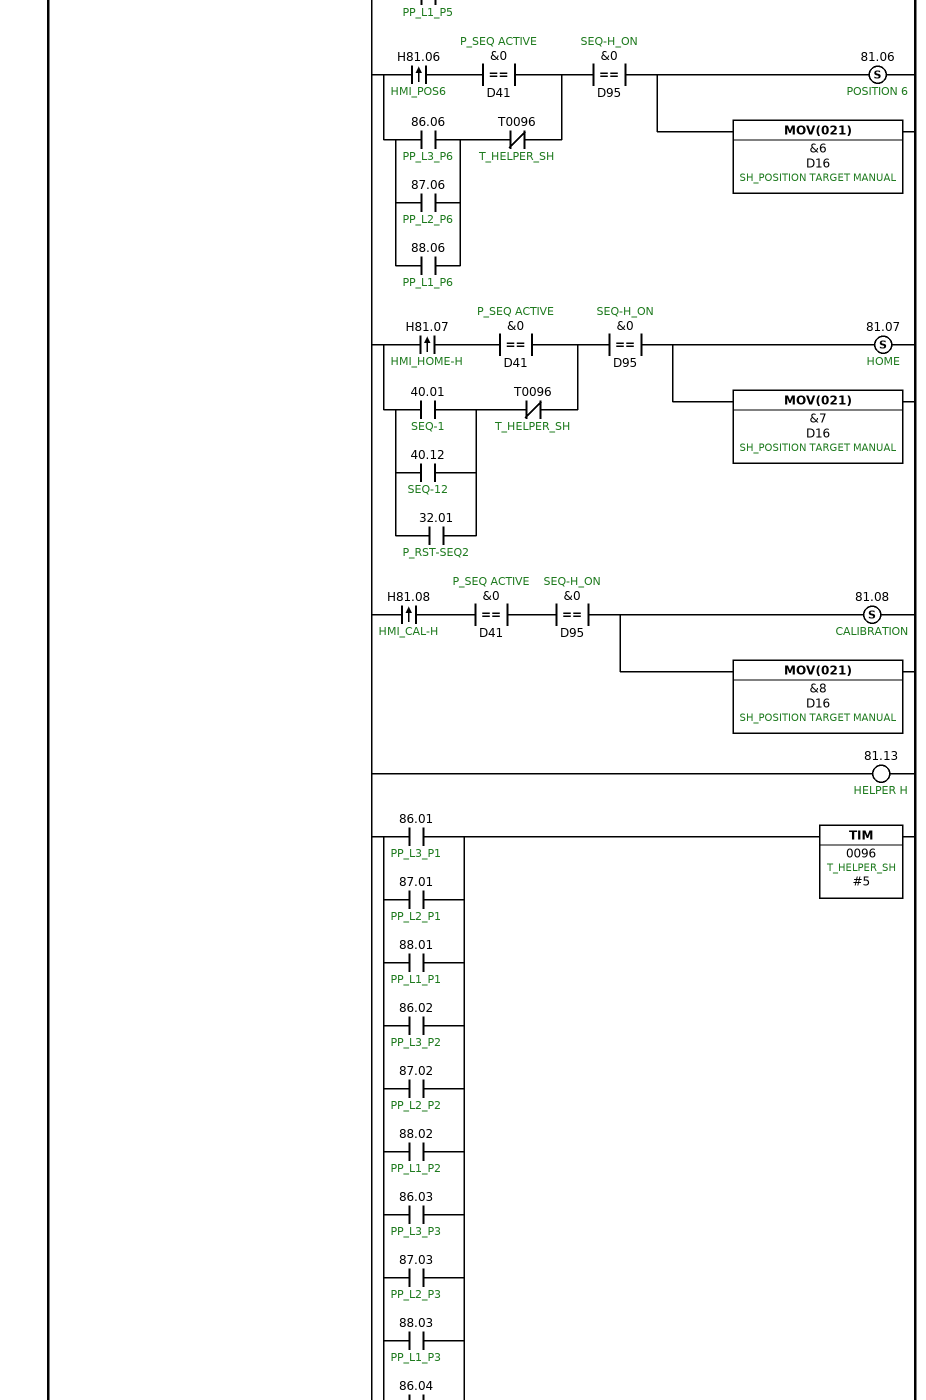
; [picture p24: NewProgram1 / SEQ_HORIZONTAL, rungs 1-1]

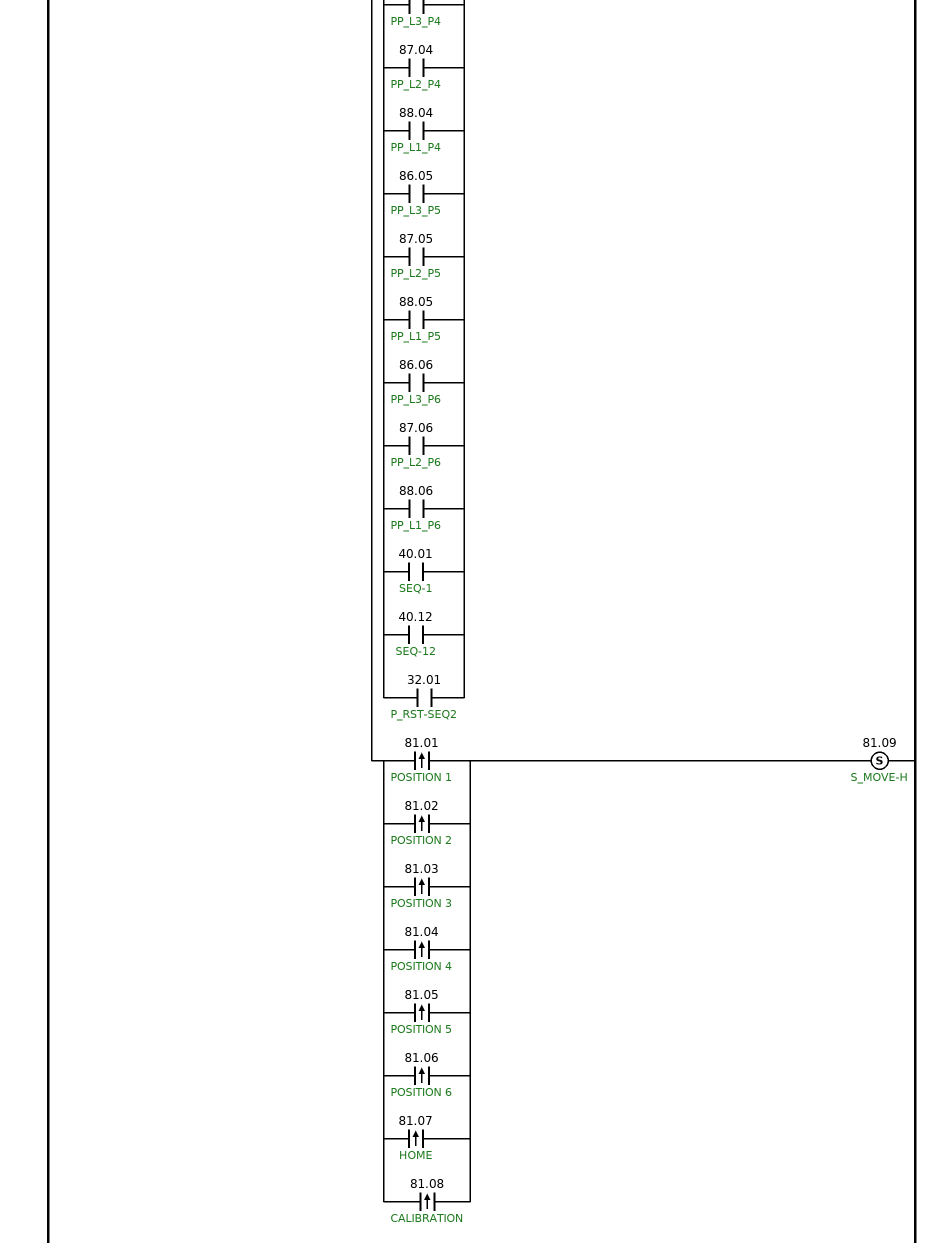
; rung 1: SET HORIZONTAL
LD P_On
LD=(300) &1 D41  ; P_SEQ ACTIVE
LD 40.01  ; SEQ-1
OR 40.08  ; SEQ-8
OR 40.12  ; SEQ-12
ANDLD
LD=(300) &1 D42  ; P_RST-SEQ_ACTIVE
AND 32.01  ; P_RST-SEQ2
ORLD
LD H30.00  ; HMI_C_MANUAL PAGE
AND=(300) &0 D41  ; P_SEQ ACTIVE
ORLD
ANDLD
OUT TR0
@LD H81.01  ; HMI_POS1
AND=(300) &0 D41  ; P_SEQ ACTIVE
LD 86.01  ; PP_L3_P1
OR 87.01  ; PP_L2_P1
OR 88.01  ; PP_L1_P1
ANDNOT T0096  ; T_HELPER_SH
ORLD
ANDLD
AND=(300) &0 D95  ; SEQ-H_ON
SET 81.01  ; POSITION 1
MOV(021) &1 D16  ; SH_POSITION TARGET MANUAL
LD TR0
@LD H81.02  ; HMI_POS2
AND=(300) &0 D41  ; P_SEQ ACTIVE
LD 86.02  ; PP_L3_P2
OR 87.02  ; PP_L2_P2
OR 88.02  ; PP_L1_P2
ANDNOT T0096  ; T_HELPER_SH
ORLD
ANDLD
AND=(300) &0 D95  ; SEQ-H_ON
SET 81.02  ; POSITION 2
MOV(021) &2 D16  ; SH_POSITION TARGET MANUAL
LD TR0
@LD H81.03  ; HMI_POS3
AND=(300) &0 D41  ; P_SEQ ACTIVE
LD 86.03  ; PP_L3_P3
OR 87.03  ; PP_L2_P3
OR 88.03  ; PP_L1_P3
ANDNOT T0096  ; T_HELPER_SH
ORLD
ANDLD
AND=(300) &0 D95  ; SEQ-H_ON
SET 81.03  ; POSITION 3
MOV(021) &3 D16  ; SH_POSITION TARGET MANUAL
LD TR0
@LD H81.04  ; HMI_POS4
AND=(300) &0 D41  ; P_SEQ ACTIVE
LD 86.04  ; PP_L3_P4
OR 87.04  ; PP_L2_P4
OR 88.04  ; PP_L1_P4
ANDNOT T0096  ; T_HELPER_SH
ORLD
ANDLD
AND=(300) &0 D95  ; SEQ-H_ON
SET 81.04  ; POSITION 4
MOV(021) &4 D16  ; SH_POSITION TARGET MANUAL
LD TR0
@LD H81.05  ; HMI_POS5
AND=(300) &0 D41  ; P_SEQ ACTIVE
LD 86.05  ; PP_L3_P5
OR 87.05  ; PP_L2_P5
OR 88.05  ; PP_L1_P5
ANDNOT T0096  ; T_HELPER_SH
ORLD
ANDLD
AND=(300) &0 D95  ; SEQ-H_ON
SET 81.05  ; POSITION 5
MOV(021) &5 D16  ; SH_POSITION TARGET MANUAL
LD TR0
@LD H81.06  ; HMI_POS6
AND=(300) &0 D41  ; P_SEQ ACTIVE
LD 86.06  ; PP_L3_P6
OR 87.06  ; PP_L2_P6
OR 88.06  ; PP_L1_P6
ANDNOT T0096  ; T_HELPER_SH
ORLD
ANDLD
AND=(300) &0 D95  ; SEQ-H_ON
SET 81.06  ; POSITION 6
MOV(021) &6 D16  ; SH_POSITION TARGET MANUAL
LD TR0
@LD H81.07  ; HMI_HOME-H
AND=(300) &0 D41  ; P_SEQ ACTIVE
LD 40.01  ; SEQ-1
OR 40.12  ; SEQ-12
OR 32.01  ; P_RST-SEQ2
ANDNOT T0096  ; T_HELPER_SH
ORLD
ANDLD
AND=(300) &0 D95  ; SEQ-H_ON
SET 81.07  ; HOME
MOV(021) &7 D16  ; SH_POSITION TARGET MANUAL
LD TR0
@AND H81.08  ; HMI_CAL-H
AND=(300) &0 D41  ; P_SEQ ACTIVE
AND=(300) &0 D95  ; SEQ-H_ON
SET 81.08  ; CALIBRATION
MOV(021) &8 D16  ; SH_POSITION TARGET MANUAL
LD TR0
OUT 81.13  ; HELPER H
LD 86.01  ; PP_L3_P1
OR 87.01  ; PP_L2_P1
OR 88.01  ; PP_L1_P1
OR 86.02  ; PP_L3_P2
OR 87.02  ; PP_L2_P2
OR 88.02  ; PP_L1_P2
OR 86.03  ; PP_L3_P3
OR 87.03  ; PP_L2_P3
OR 88.03  ; PP_L1_P3
OR 86.04  ; PP_L3_P4
OR 87.04  ; PP_L2_P4
OR 88.04  ; PP_L1_P4
OR 86.05  ; PP_L3_P5
OR 87.05  ; PP_L2_P5
OR 88.05  ; PP_L1_P5
OR 86.06  ; PP_L3_P6
OR 87.06  ; PP_L2_P6
OR 88.06  ; PP_L1_P6
OR 40.01  ; SEQ-1
OR 40.12  ; SEQ-12
OR 32.01  ; P_RST-SEQ2
ANDLD
TIM 0096 #5  ; T_HELPER_SH
LD TR0
@LD 81.01  ; POSITION 1
@OR 81.02  ; POSITION 2
@OR 81.03  ; POSITION 3
@OR 81.04  ; POSITION 4
@OR 81.05  ; POSITION 5
@OR 81.06  ; POSITION 6
@OR 81.07  ; HOME
@OR 81.08  ; CALIBRATION
ANDLD
SET 81.09  ; S_MOVE-H

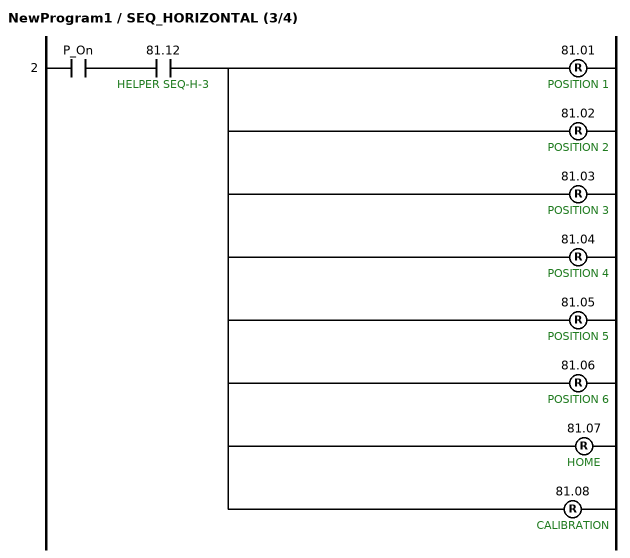
; rung 2
LD P_On
AND 81.12  ; HELPER SEQ-H-3
RSET 81.01  ; POSITION 1
RSET 81.02  ; POSITION 2
RSET 81.03  ; POSITION 3
RSET 81.04  ; POSITION 4
RSET 81.05  ; POSITION 5
RSET 81.06  ; POSITION 6
RSET 81.07  ; HOME
RSET 81.08  ; CALIBRATION

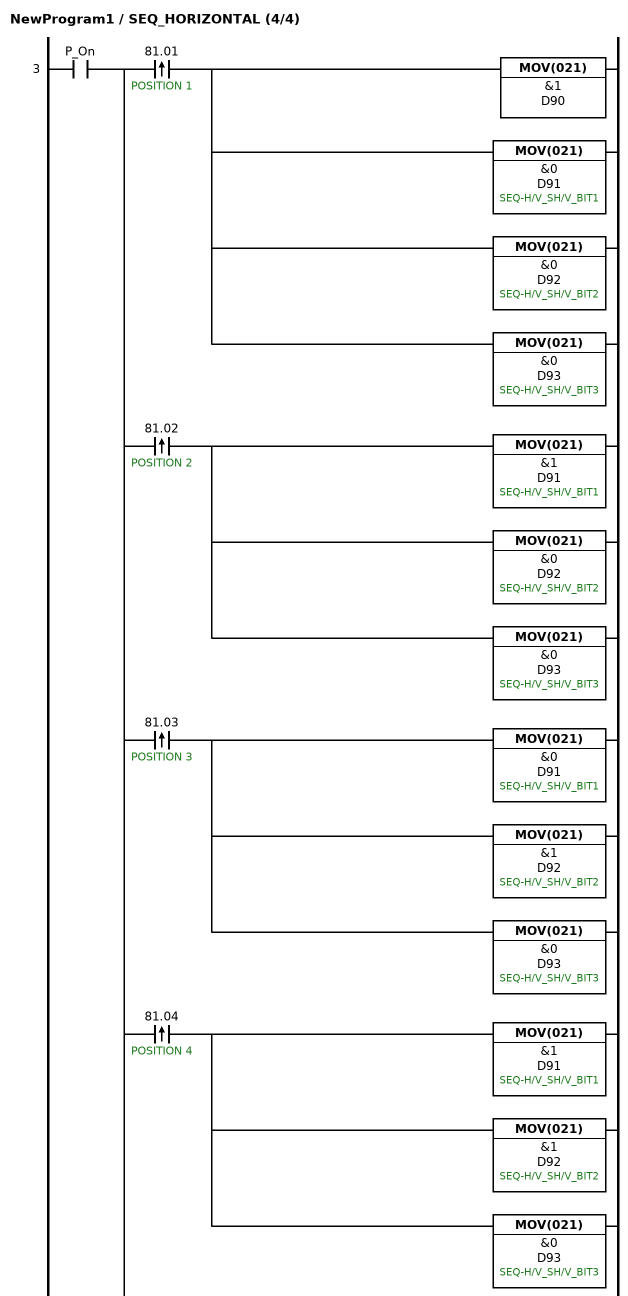

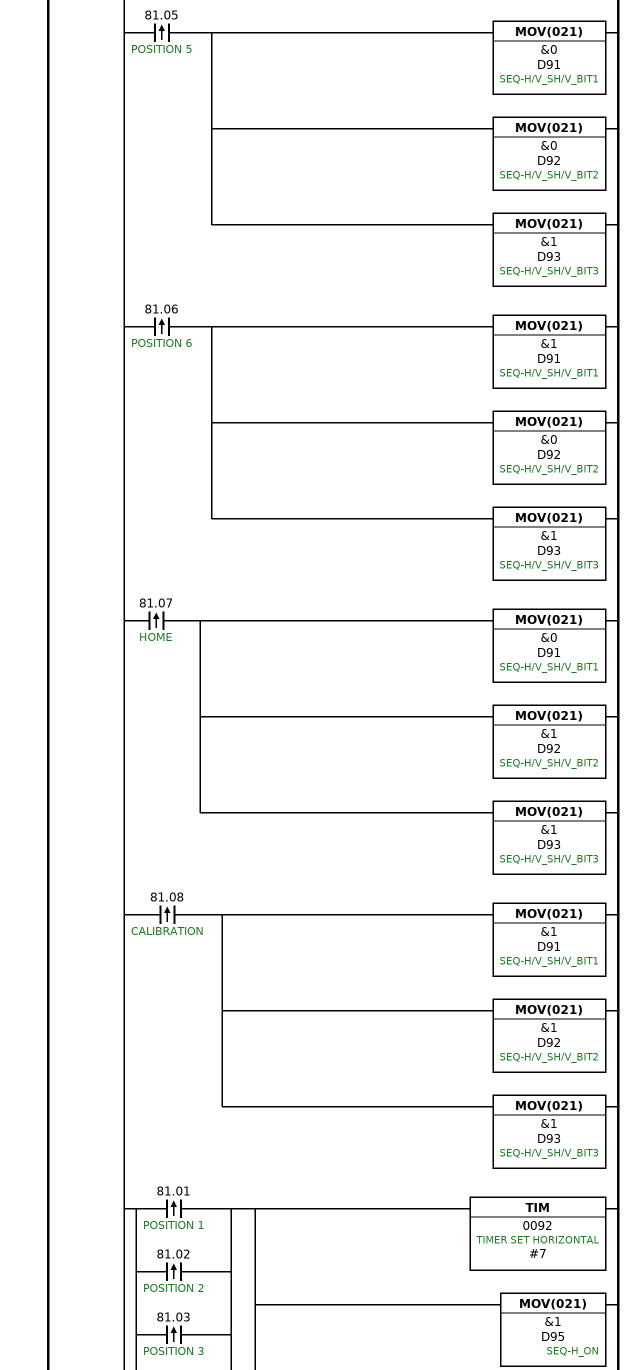

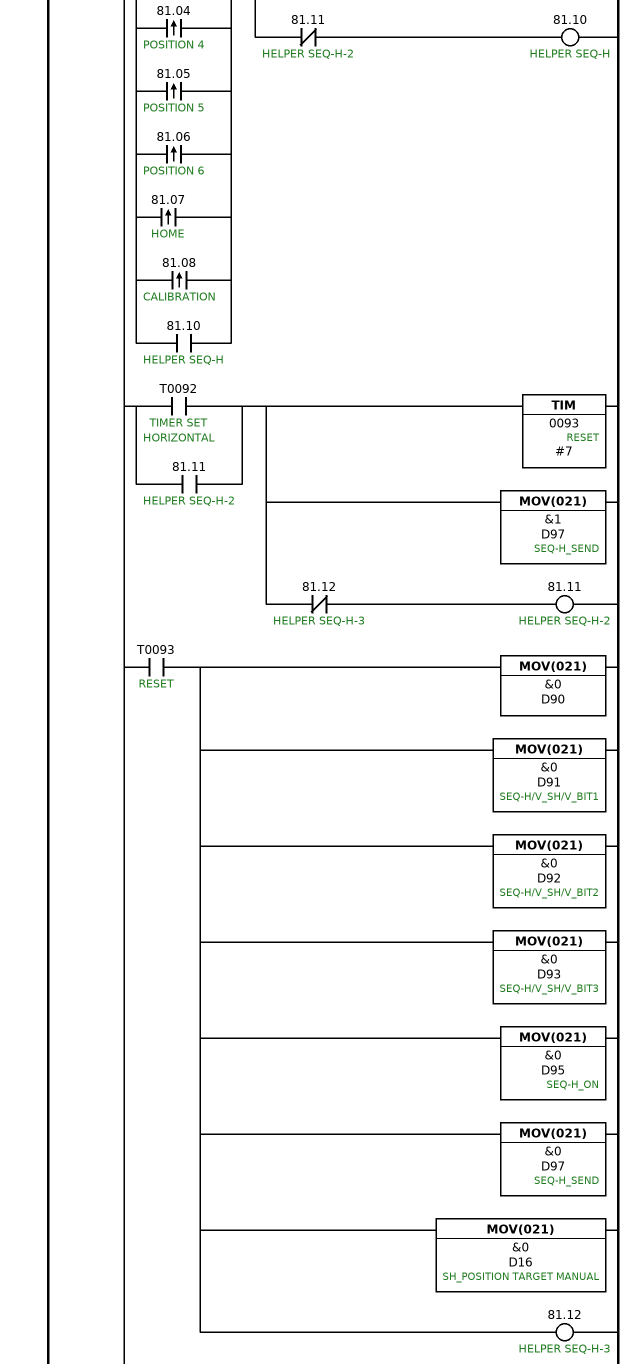

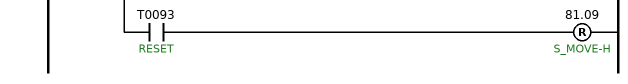
; rung 3
LD P_On
OUT TR0
@AND 81.01  ; POSITION 1
MOV(021) &1 D90
MOV(021) &0 D91  ; SEQ-H/V_SH/V_BIT1
MOV(021) &0 D92  ; SEQ-H/V_SH/V_BIT2
MOV(021) &0 D93  ; SEQ-H/V_SH/V_BIT3
LD TR0
@AND 81.02  ; POSITION 2
MOV(021) &1 D91  ; SEQ-H/V_SH/V_BIT1
MOV(021) &0 D92  ; SEQ-H/V_SH/V_BIT2
MOV(021) &0 D93  ; SEQ-H/V_SH/V_BIT3
LD TR0
@AND 81.03  ; POSITION 3
MOV(021) &0 D91  ; SEQ-H/V_SH/V_BIT1
MOV(021) &1 D92  ; SEQ-H/V_SH/V_BIT2
MOV(021) &0 D93  ; SEQ-H/V_SH/V_BIT3
LD TR0
@AND 81.04  ; POSITION 4
MOV(021) &1 D91  ; SEQ-H/V_SH/V_BIT1
MOV(021) &1 D92  ; SEQ-H/V_SH/V_BIT2
MOV(021) &0 D93  ; SEQ-H/V_SH/V_BIT3
LD TR0
@AND 81.05  ; POSITION 5
MOV(021) &0 D91  ; SEQ-H/V_SH/V_BIT1
MOV(021) &0 D92  ; SEQ-H/V_SH/V_BIT2
MOV(021) &1 D93  ; SEQ-H/V_SH/V_BIT3
LD TR0
@AND 81.06  ; POSITION 6
MOV(021) &1 D91  ; SEQ-H/V_SH/V_BIT1
MOV(021) &0 D92  ; SEQ-H/V_SH/V_BIT2
MOV(021) &1 D93  ; SEQ-H/V_SH/V_BIT3
LD TR0
@AND 81.07  ; HOME
MOV(021) &0 D91  ; SEQ-H/V_SH/V_BIT1
MOV(021) &1 D92  ; SEQ-H/V_SH/V_BIT2
MOV(021) &1 D93  ; SEQ-H/V_SH/V_BIT3
LD TR0
@AND 81.08  ; CALIBRATION
MOV(021) &1 D91  ; SEQ-H/V_SH/V_BIT1
MOV(021) &1 D92  ; SEQ-H/V_SH/V_BIT2
MOV(021) &1 D93  ; SEQ-H/V_SH/V_BIT3
LD TR0
@LD 81.01  ; POSITION 1
@OR 81.02  ; POSITION 2
@OR 81.03  ; POSITION 3
@OR 81.04  ; POSITION 4
@OR 81.05  ; POSITION 5
@OR 81.06  ; POSITION 6
@OR 81.07  ; HOME
@OR 81.08  ; CALIBRATION
OR 81.10  ; HELPER SEQ-H
ANDLD
TIM 0092 #7  ; TIMER SET HORIZONTAL
MOV(021) &1 D95  ; SEQ-H_ON
ANDNOT 81.11  ; HELPER SEQ-H-2
OUT 81.10  ; HELPER SEQ-H
LD TR0
LD T0092  ; TIMER SET HORIZONTAL
OR 81.11  ; HELPER SEQ-H-2
ANDLD
TIM 0093 #7  ; RESET
MOV(021) &1 D97  ; SEQ-H_SEND
ANDNOT 81.12  ; HELPER SEQ-H-3
OUT 81.11  ; HELPER SEQ-H-2
LD TR0
AND T0093  ; RESET
MOV(021) &0 D90
MOV(021) &0 D91  ; SEQ-H/V_SH/V_BIT1
MOV(021) &0 D92  ; SEQ-H/V_SH/V_BIT2
MOV(021) &0 D93  ; SEQ-H/V_SH/V_BIT3
MOV(021) &0 D95  ; SEQ-H_ON
MOV(021) &0 D97  ; SEQ-H_SEND
MOV(021) &0 D16  ; SH_POSITION TARGET MANUAL
OUT 81.12  ; HELPER SEQ-H-3
LD TR0
AND T0093  ; RESET
RSET 81.09  ; S_MOVE-H

### Section SEQ_VERTICAL

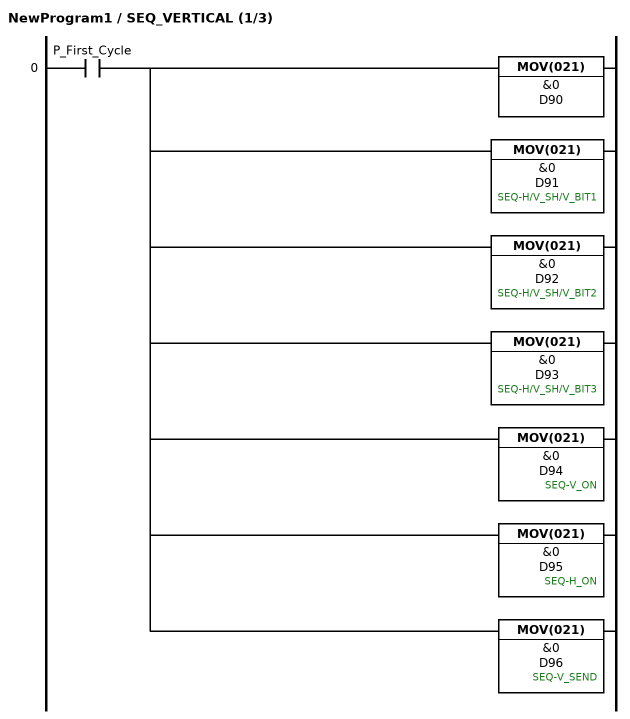
; rung 0
LD P_First_Cycle
MOV(021) &0 D90
MOV(021) &0 D91  ; SEQ-H/V_SH/V_BIT1
MOV(021) &0 D92  ; SEQ-H/V_SH/V_BIT2
MOV(021) &0 D93  ; SEQ-H/V_SH/V_BIT3
MOV(021) &0 D94  ; SEQ-V_ON
MOV(021) &0 D95  ; SEQ-H_ON
MOV(021) &0 D96  ; SEQ-V_SEND

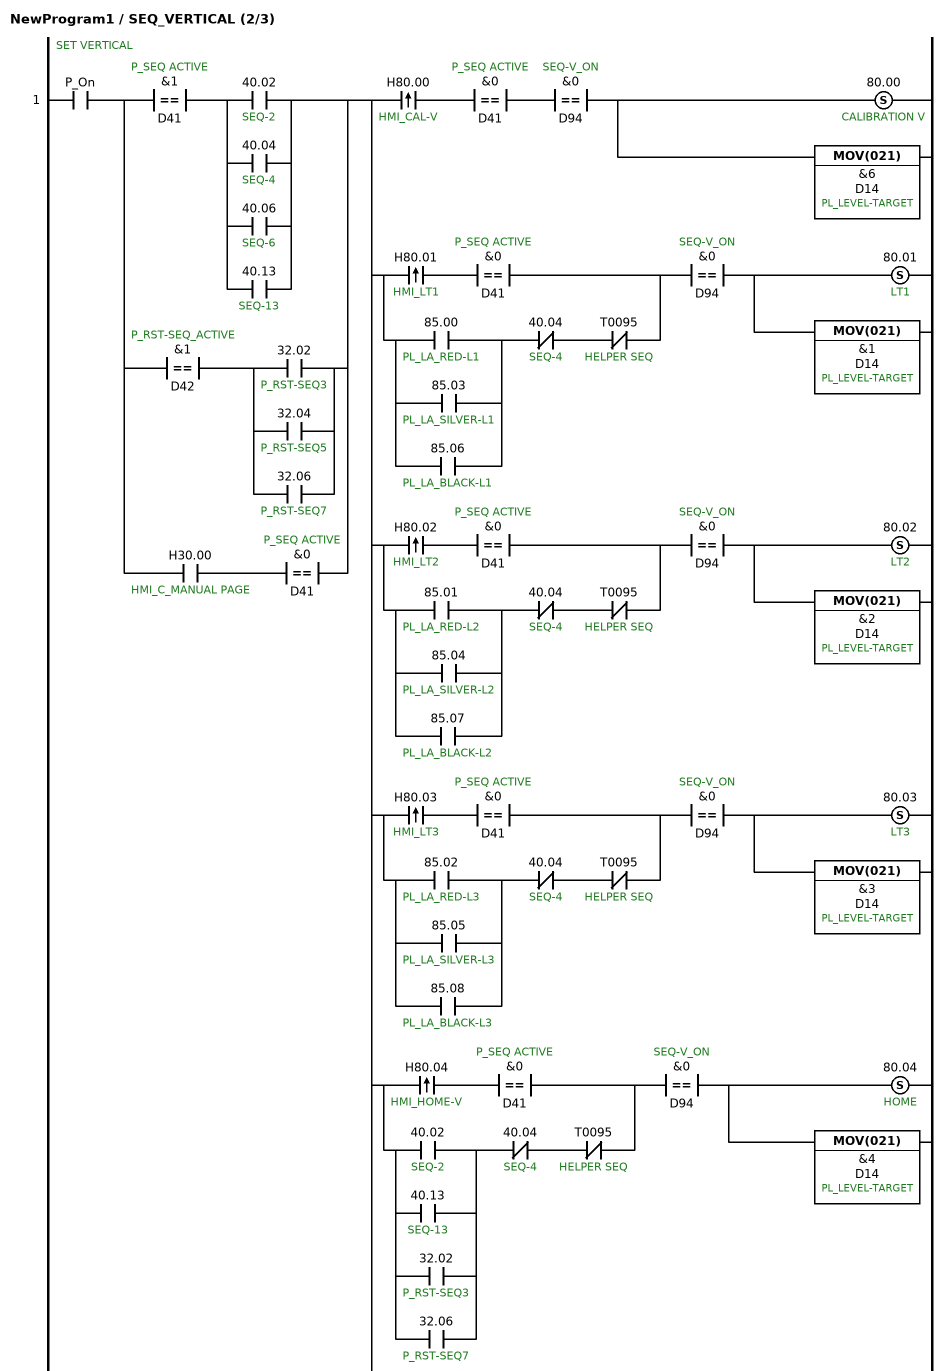

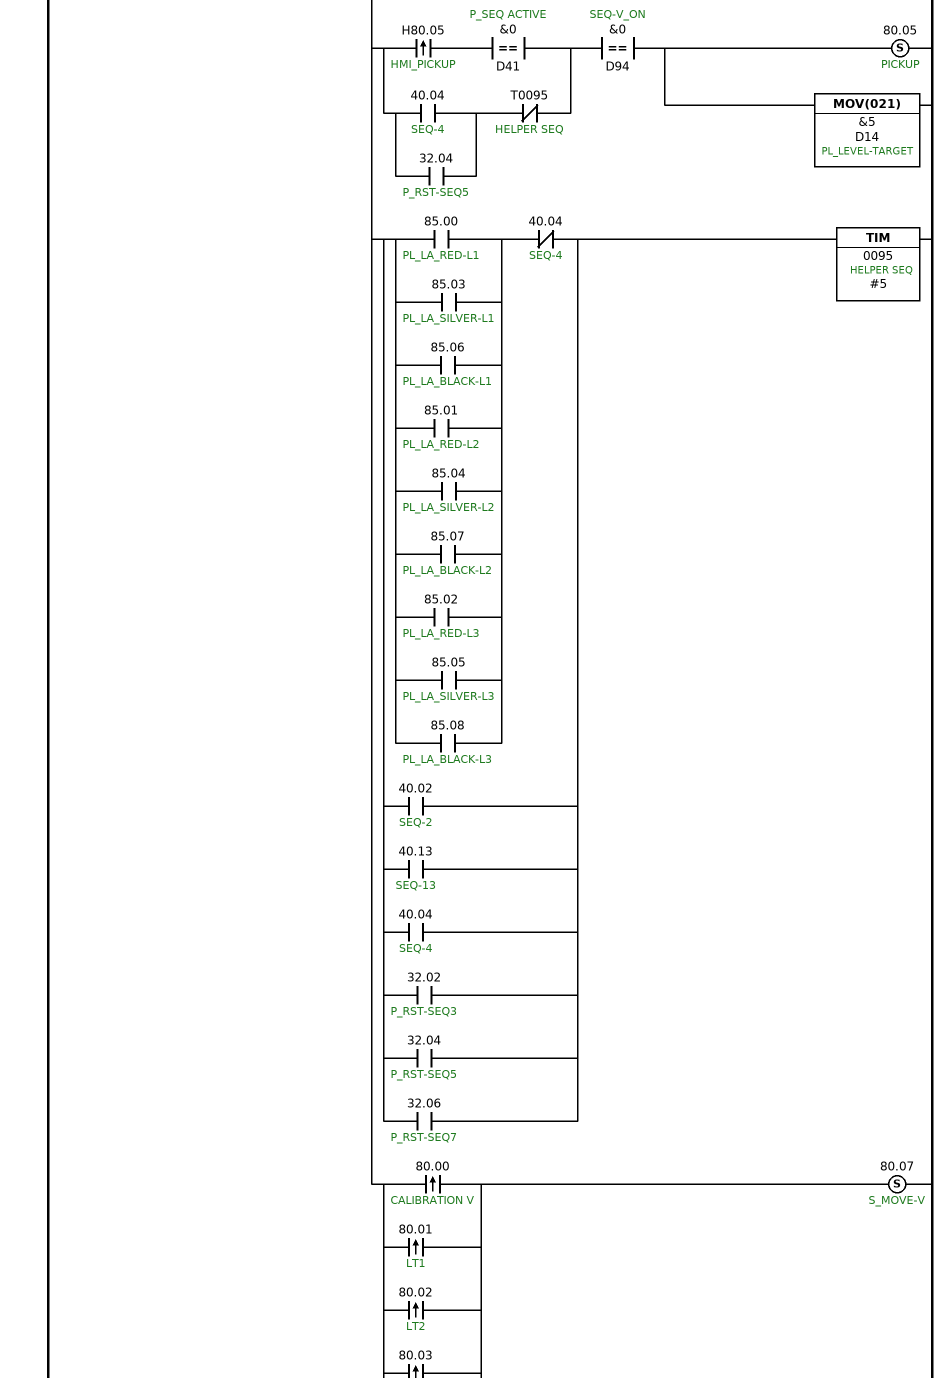

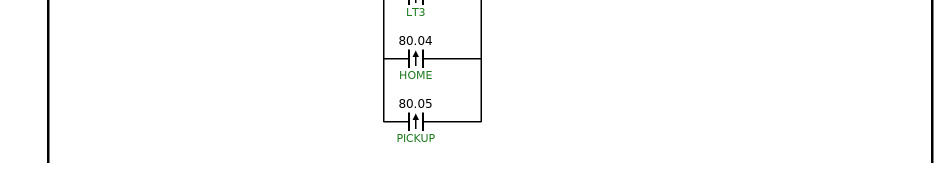
; rung 1: SET VERTICAL
LD P_On
LD=(300) &1 D41  ; P_SEQ ACTIVE
LD 40.02  ; SEQ-2
OR 40.04  ; SEQ-4
OR 40.06  ; SEQ-6
OR 40.13  ; SEQ-13
ANDLD
LD=(300) &1 D42  ; P_RST-SEQ_ACTIVE
LD 32.02  ; P_RST-SEQ3
OR 32.04  ; P_RST-SEQ5
OR 32.06  ; P_RST-SEQ7
ANDLD
ORLD
LD H30.00  ; HMI_C_MANUAL PAGE
AND=(300) &0 D41  ; P_SEQ ACTIVE
ORLD
ANDLD
OUT TR0
@AND H80.00  ; HMI_CAL-V
AND=(300) &0 D41  ; P_SEQ ACTIVE
AND=(300) &0 D94  ; SEQ-V_ON
SET 80.00  ; CALIBRATION V
MOV(021) &6 D14  ; PL_LEVEL-TARGET
LD TR0
@LD H80.01  ; HMI_LT1
AND=(300) &0 D41  ; P_SEQ ACTIVE
LD 85.00  ; PL_LA_RED-L1
OR 85.03  ; PL_LA_SILVER-L1
OR 85.06  ; PL_LA_BLACK-L1
ANDNOT 40.04  ; SEQ-4
ANDNOT T0095  ; HELPER SEQ
ORLD
ANDLD
AND=(300) &0 D94  ; SEQ-V_ON
SET 80.01  ; LT1
MOV(021) &1 D14  ; PL_LEVEL-TARGET
LD TR0
@LD H80.02  ; HMI_LT2
AND=(300) &0 D41  ; P_SEQ ACTIVE
LD 85.01  ; PL_LA_RED-L2
OR 85.04  ; PL_LA_SILVER-L2
OR 85.07  ; PL_LA_BLACK-L2
ANDNOT 40.04  ; SEQ-4
ANDNOT T0095  ; HELPER SEQ
ORLD
ANDLD
AND=(300) &0 D94  ; SEQ-V_ON
SET 80.02  ; LT2
MOV(021) &2 D14  ; PL_LEVEL-TARGET
LD TR0
@LD H80.03  ; HMI_LT3
AND=(300) &0 D41  ; P_SEQ ACTIVE
LD 85.02  ; PL_LA_RED-L3
OR 85.05  ; PL_LA_SILVER-L3
OR 85.08  ; PL_LA_BLACK-L3
ANDNOT 40.04  ; SEQ-4
ANDNOT T0095  ; HELPER SEQ
ORLD
ANDLD
AND=(300) &0 D94  ; SEQ-V_ON
SET 80.03  ; LT3
MOV(021) &3 D14  ; PL_LEVEL-TARGET
LD TR0
@LD H80.04  ; HMI_HOME-V
AND=(300) &0 D41  ; P_SEQ ACTIVE
LD 40.02  ; SEQ-2
OR 40.13  ; SEQ-13
OR 32.02  ; P_RST-SEQ3
OR 32.06  ; P_RST-SEQ7
ANDNOT 40.04  ; SEQ-4
ANDNOT T0095  ; HELPER SEQ
ORLD
ANDLD
AND=(300) &0 D94  ; SEQ-V_ON
SET 80.04  ; HOME
MOV(021) &4 D14  ; PL_LEVEL-TARGET
LD TR0
@LD H80.05  ; HMI_PICKUP
AND=(300) &0 D41  ; P_SEQ ACTIVE
LD 40.04  ; SEQ-4
OR 32.04  ; P_RST-SEQ5
ANDNOT T0095  ; HELPER SEQ
ORLD
ANDLD
AND=(300) &0 D94  ; SEQ-V_ON
SET 80.05  ; PICKUP
MOV(021) &5 D14  ; PL_LEVEL-TARGET
LD TR0
LD 85.00  ; PL_LA_RED-L1
OR 85.03  ; PL_LA_SILVER-L1
OR 85.06  ; PL_LA_BLACK-L1
OR 85.01  ; PL_LA_RED-L2
OR 85.04  ; PL_LA_SILVER-L2
OR 85.07  ; PL_LA_BLACK-L2
OR 85.02  ; PL_LA_RED-L3
OR 85.05  ; PL_LA_SILVER-L3
OR 85.08  ; PL_LA_BLACK-L3
ANDNOT 40.04  ; SEQ-4
OR 40.02  ; SEQ-2
OR 40.13  ; SEQ-13
OR 40.04  ; SEQ-4
OR 32.02  ; P_RST-SEQ3
OR 32.04  ; P_RST-SEQ5
OR 32.06  ; P_RST-SEQ7
ANDLD
TIM 0095 #5  ; HELPER SEQ
LD TR0
@LD 80.00  ; CALIBRATION V
@OR 80.01  ; LT1
@OR 80.02  ; LT2
@OR 80.03  ; LT3
@OR 80.04  ; HOME
@OR 80.05  ; PICKUP
ANDLD
SET 80.07  ; S_MOVE-V

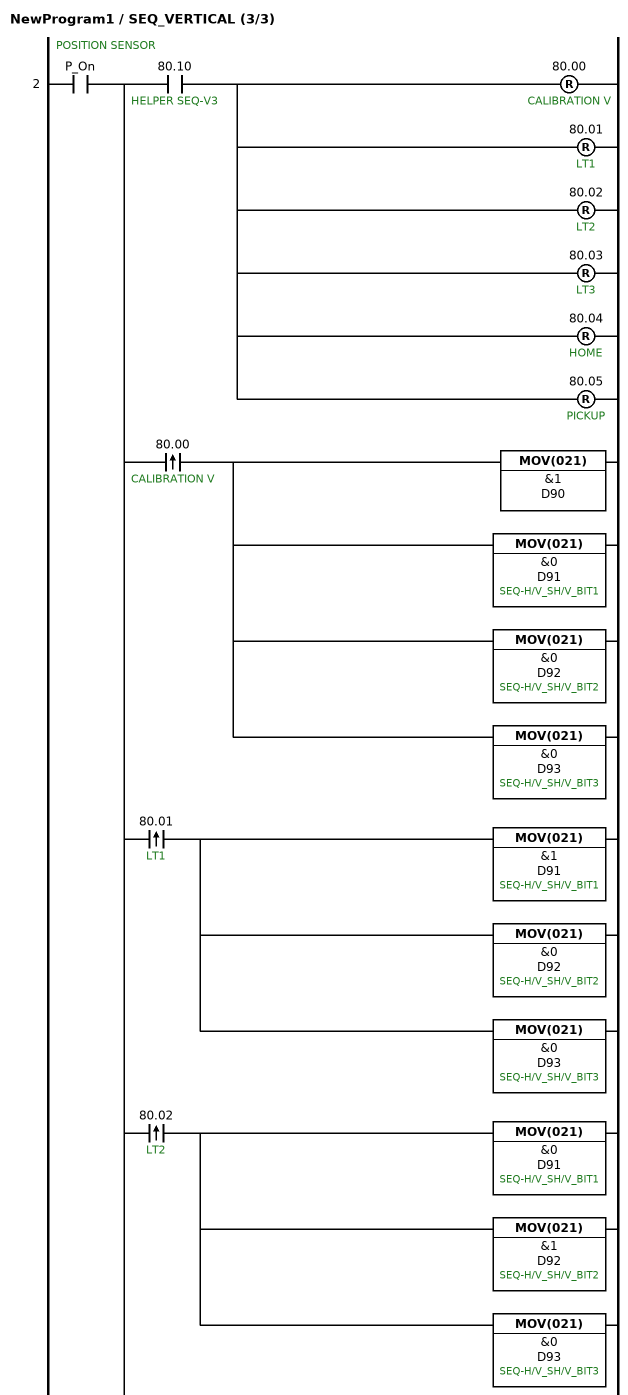

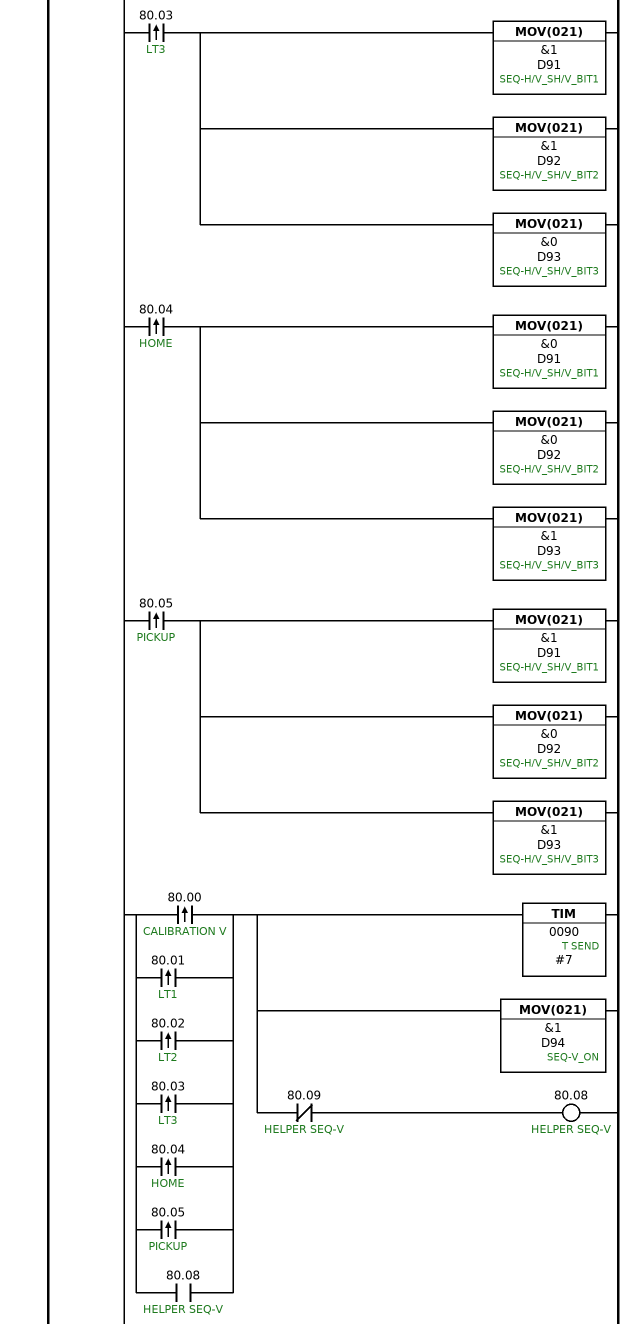

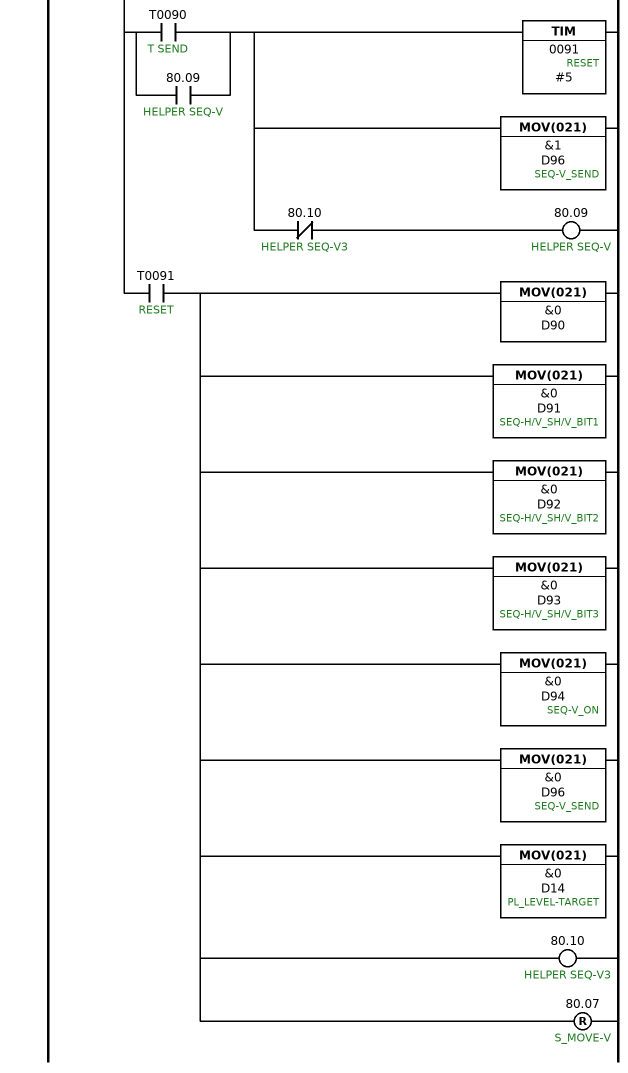
; rung 2: POSITION SENSOR
LD P_On
OUT TR0
AND 80.10  ; HELPER SEQ-V3
RSET 80.00  ; CALIBRATION V
RSET 80.01  ; LT1
RSET 80.02  ; LT2
RSET 80.03  ; LT3
RSET 80.04  ; HOME
RSET 80.05  ; PICKUP
LD TR0
@AND 80.00  ; CALIBRATION V
MOV(021) &1 D90
MOV(021) &0 D91  ; SEQ-H/V_SH/V_BIT1
MOV(021) &0 D92  ; SEQ-H/V_SH/V_BIT2
MOV(021) &0 D93  ; SEQ-H/V_SH/V_BIT3
LD TR0
@AND 80.01  ; LT1
MOV(021) &1 D91  ; SEQ-H/V_SH/V_BIT1
MOV(021) &0 D92  ; SEQ-H/V_SH/V_BIT2
MOV(021) &0 D93  ; SEQ-H/V_SH/V_BIT3
LD TR0
@AND 80.02  ; LT2
MOV(021) &0 D91  ; SEQ-H/V_SH/V_BIT1
MOV(021) &1 D92  ; SEQ-H/V_SH/V_BIT2
MOV(021) &0 D93  ; SEQ-H/V_SH/V_BIT3
LD TR0
@AND 80.03  ; LT3
MOV(021) &1 D91  ; SEQ-H/V_SH/V_BIT1
MOV(021) &1 D92  ; SEQ-H/V_SH/V_BIT2
MOV(021) &0 D93  ; SEQ-H/V_SH/V_BIT3
LD TR0
@AND 80.04  ; HOME
MOV(021) &0 D91  ; SEQ-H/V_SH/V_BIT1
MOV(021) &0 D92  ; SEQ-H/V_SH/V_BIT2
MOV(021) &1 D93  ; SEQ-H/V_SH/V_BIT3
LD TR0
@AND 80.05  ; PICKUP
MOV(021) &1 D91  ; SEQ-H/V_SH/V_BIT1
MOV(021) &0 D92  ; SEQ-H/V_SH/V_BIT2
MOV(021) &1 D93  ; SEQ-H/V_SH/V_BIT3
LD TR0
@LD 80.00  ; CALIBRATION V
@OR 80.01  ; LT1
@OR 80.02  ; LT2
@OR 80.03  ; LT3
@OR 80.04  ; HOME
@OR 80.05  ; PICKUP
OR 80.08  ; HELPER SEQ-V
ANDLD
TIM 0090 #7  ; T SEND
MOV(021) &1 D94  ; SEQ-V_ON
ANDNOT 80.09  ; HELPER SEQ-V
OUT 80.08  ; HELPER SEQ-V
LD TR0
LD T0090  ; T SEND
OR 80.09  ; HELPER SEQ-V
ANDLD
TIM 0091 #5  ; RESET
MOV(021) &1 D96  ; SEQ-V_SEND
ANDNOT 80.10  ; HELPER SEQ-V3
OUT 80.09  ; HELPER SEQ-V
LD TR0
AND T0091  ; RESET
MOV(021) &0 D90
MOV(021) &0 D91  ; SEQ-H/V_SH/V_BIT1
MOV(021) &0 D92  ; SEQ-H/V_SH/V_BIT2
MOV(021) &0 D93  ; SEQ-H/V_SH/V_BIT3
MOV(021) &0 D94  ; SEQ-V_ON
MOV(021) &0 D96  ; SEQ-V_SEND
MOV(021) &0 D14  ; PL_LEVEL-TARGET
OUT 80.10  ; HELPER SEQ-V3
RSET 80.07  ; S_MOVE-V

### Section SEQUENCE

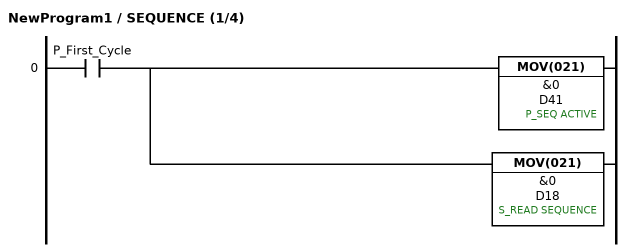
; rung 0
LD P_First_Cycle
MOV(021) &0 D41  ; P_SEQ ACTIVE
MOV(021) &0 D18  ; S_READ SEQUENCE

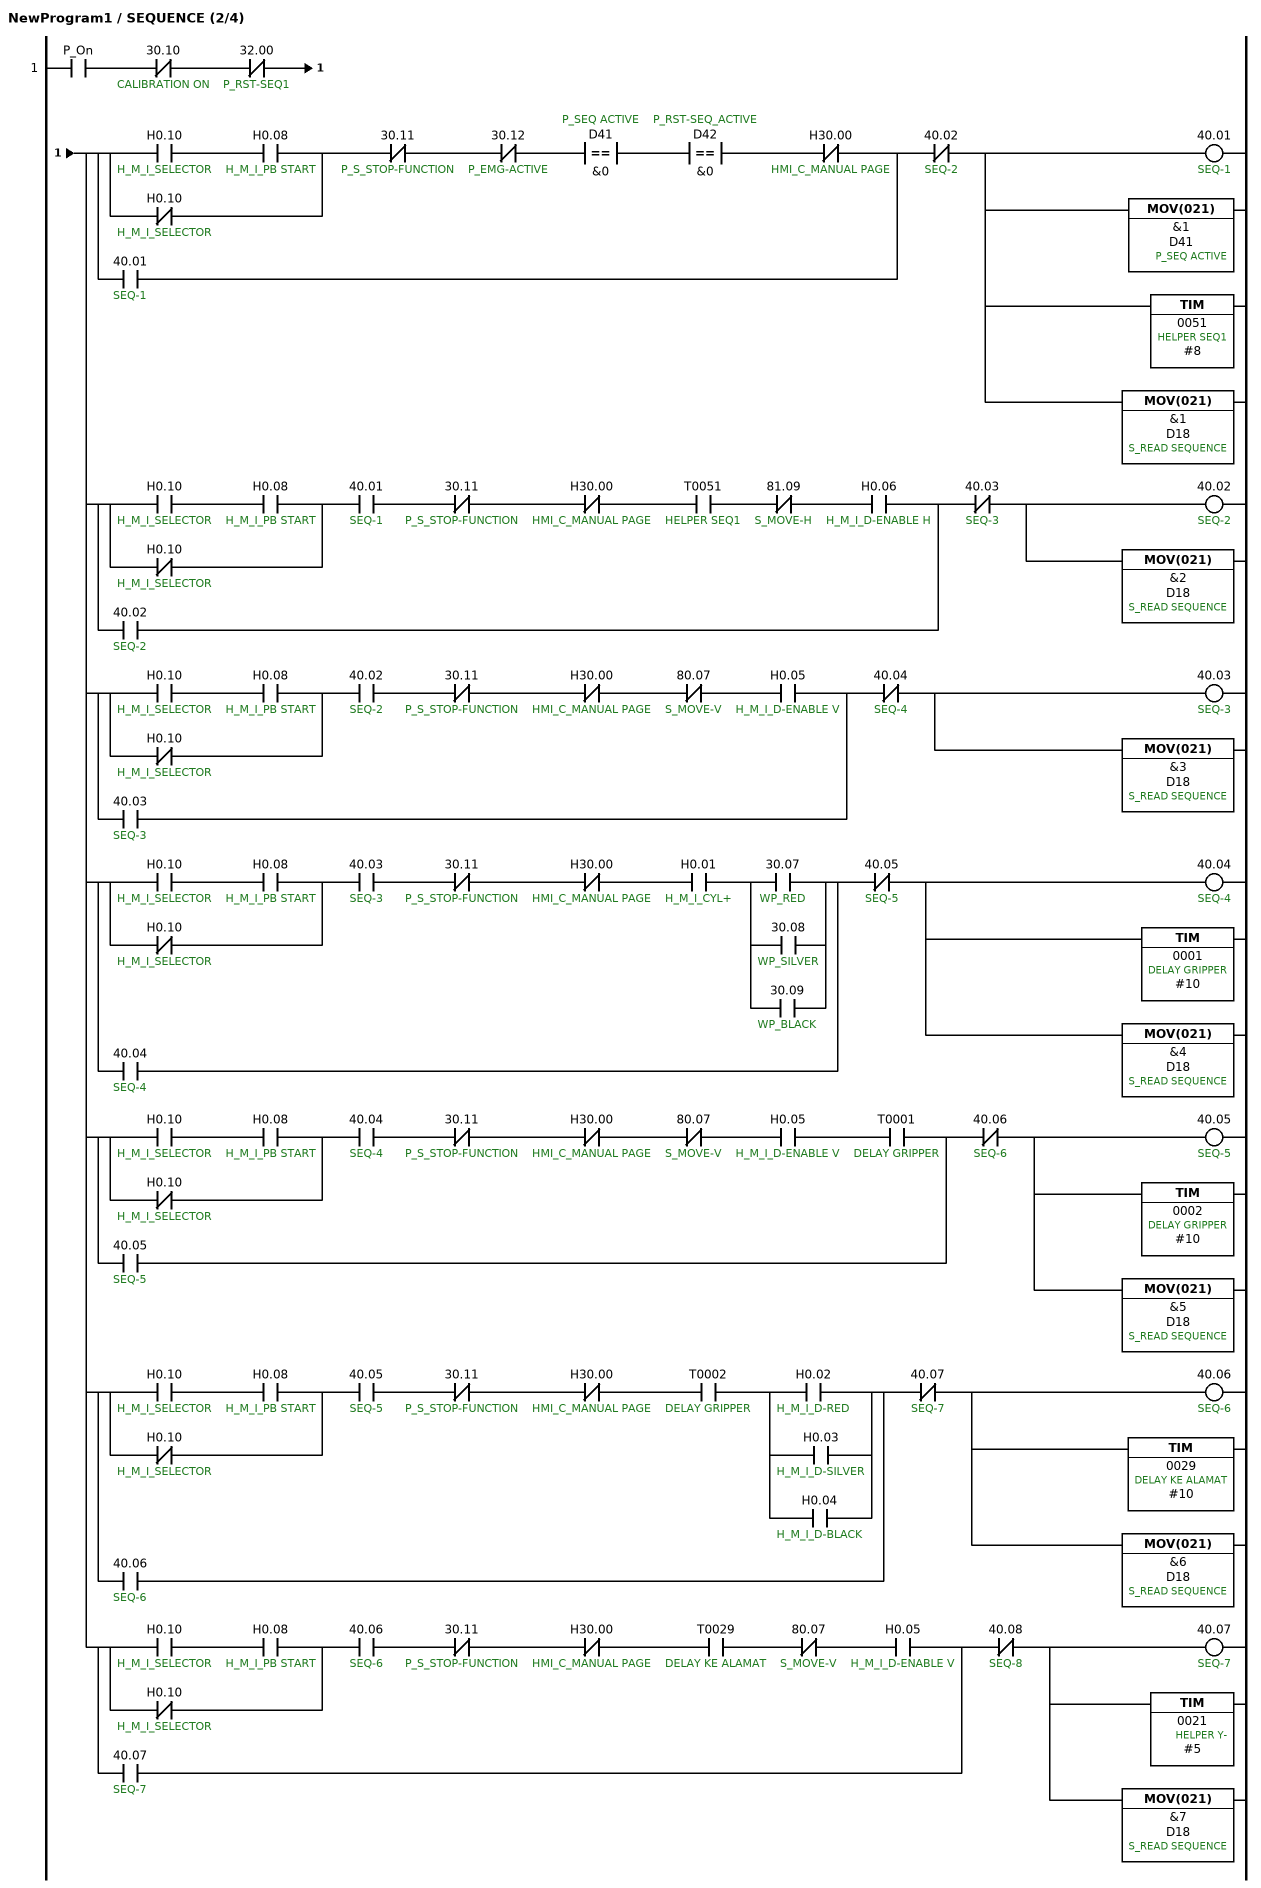
; rung 1
LD P_On
ANDNOT 30.10  ; CALIBRATION ON
ANDNOT 32.00  ; P_RST-SEQ1
OUT TR0
LD H0.10  ; H_M_I_SELECTOR
AND H0.08  ; H_M_I_PB START
ORNOT H0.10  ; H_M_I_SELECTOR
ANDNOT 30.11  ; P_S_STOP-FUNCTION
ANDNOT 30.12  ; P_EMG-ACTIVE
AND=(300) D41 &0  ; P_SEQ ACTIVE
AND=(300) D42 &0  ; P_RST-SEQ_ACTIVE
ANDNOT H30.00  ; HMI_C_MANUAL PAGE
OR 40.01  ; SEQ-1
ANDLD
ANDNOT 40.02  ; SEQ-2
OUT 40.01  ; SEQ-1
MOV(021) &1 D41  ; P_SEQ ACTIVE
TIM 0051 #8  ; HELPER SEQ1
MOV(021) &1 D18  ; S_READ SEQUENCE
LD TR0
LD H0.10  ; H_M_I_SELECTOR
AND H0.08  ; H_M_I_PB START
ORNOT H0.10  ; H_M_I_SELECTOR
AND 40.01  ; SEQ-1
ANDNOT 30.11  ; P_S_STOP-FUNCTION
ANDNOT H30.00  ; HMI_C_MANUAL PAGE
AND T0051  ; HELPER SEQ1
ANDNOT 81.09  ; S_MOVE-H
AND H0.06  ; H_M_I_D-ENABLE H
OR 40.02  ; SEQ-2
ANDLD
ANDNOT 40.03  ; SEQ-3
OUT 40.02  ; SEQ-2
MOV(021) &2 D18  ; S_READ SEQUENCE
LD TR0
LD H0.10  ; H_M_I_SELECTOR
AND H0.08  ; H_M_I_PB START
ORNOT H0.10  ; H_M_I_SELECTOR
AND 40.02  ; SEQ-2
ANDNOT 30.11  ; P_S_STOP-FUNCTION
ANDNOT H30.00  ; HMI_C_MANUAL PAGE
ANDNOT 80.07  ; S_MOVE-V
AND H0.05  ; H_M_I_D-ENABLE V
OR 40.03  ; SEQ-3
ANDLD
ANDNOT 40.04  ; SEQ-4
OUT 40.03  ; SEQ-3
MOV(021) &3 D18  ; S_READ SEQUENCE
LD TR0
LD H0.10  ; H_M_I_SELECTOR
AND H0.08  ; H_M_I_PB START
ORNOT H0.10  ; H_M_I_SELECTOR
AND 40.03  ; SEQ-3
ANDNOT 30.11  ; P_S_STOP-FUNCTION
ANDNOT H30.00  ; HMI_C_MANUAL PAGE
AND H0.01  ; H_M_I_CYL+
LD 30.07  ; WP_RED
OR 30.08  ; WP_SILVER
OR 30.09  ; WP_BLACK
ANDLD
OR 40.04  ; SEQ-4
ANDLD
ANDNOT 40.05  ; SEQ-5
OUT 40.04  ; SEQ-4
TIM 0001 #10  ; DELAY GRIPPER
MOV(021) &4 D18  ; S_READ SEQUENCE
LD TR0
LD H0.10  ; H_M_I_SELECTOR
AND H0.08  ; H_M_I_PB START
ORNOT H0.10  ; H_M_I_SELECTOR
AND 40.04  ; SEQ-4
ANDNOT 30.11  ; P_S_STOP-FUNCTION
ANDNOT H30.00  ; HMI_C_MANUAL PAGE
ANDNOT 80.07  ; S_MOVE-V
AND H0.05  ; H_M_I_D-ENABLE V
AND T0001  ; DELAY GRIPPER
OR 40.05  ; SEQ-5
ANDLD
ANDNOT 40.06  ; SEQ-6
OUT 40.05  ; SEQ-5
TIM 0002 #10  ; DELAY GRIPPER
MOV(021) &5 D18  ; S_READ SEQUENCE
LD TR0
LD H0.10  ; H_M_I_SELECTOR
AND H0.08  ; H_M_I_PB START
ORNOT H0.10  ; H_M_I_SELECTOR
AND 40.05  ; SEQ-5
ANDNOT 30.11  ; P_S_STOP-FUNCTION
ANDNOT H30.00  ; HMI_C_MANUAL PAGE
AND T0002  ; DELAY GRIPPER
LD H0.02  ; H_M_I_D-RED
OR H0.03  ; H_M_I_D-SILVER
OR H0.04  ; H_M_I_D-BLACK
ANDLD
OR 40.06  ; SEQ-6
ANDLD
ANDNOT 40.07  ; SEQ-7
OUT 40.06  ; SEQ-6
TIM 0029 #10  ; DELAY KE ALAMAT
MOV(021) &6 D18  ; S_READ SEQUENCE
LD TR0
LD H0.10  ; H_M_I_SELECTOR
AND H0.08  ; H_M_I_PB START
ORNOT H0.10  ; H_M_I_SELECTOR
AND 40.06  ; SEQ-6
ANDNOT 30.11  ; P_S_STOP-FUNCTION
ANDNOT H30.00  ; HMI_C_MANUAL PAGE
AND T0029  ; DELAY KE ALAMAT
ANDNOT 80.07  ; S_MOVE-V
AND H0.05  ; H_M_I_D-ENABLE V
OR 40.07  ; SEQ-7
ANDLD
ANDNOT 40.08  ; SEQ-8
OUT 40.07  ; SEQ-7
TIM 0021 #5  ; HELPER Y-
MOV(021) &7 D18  ; S_READ SEQUENCE

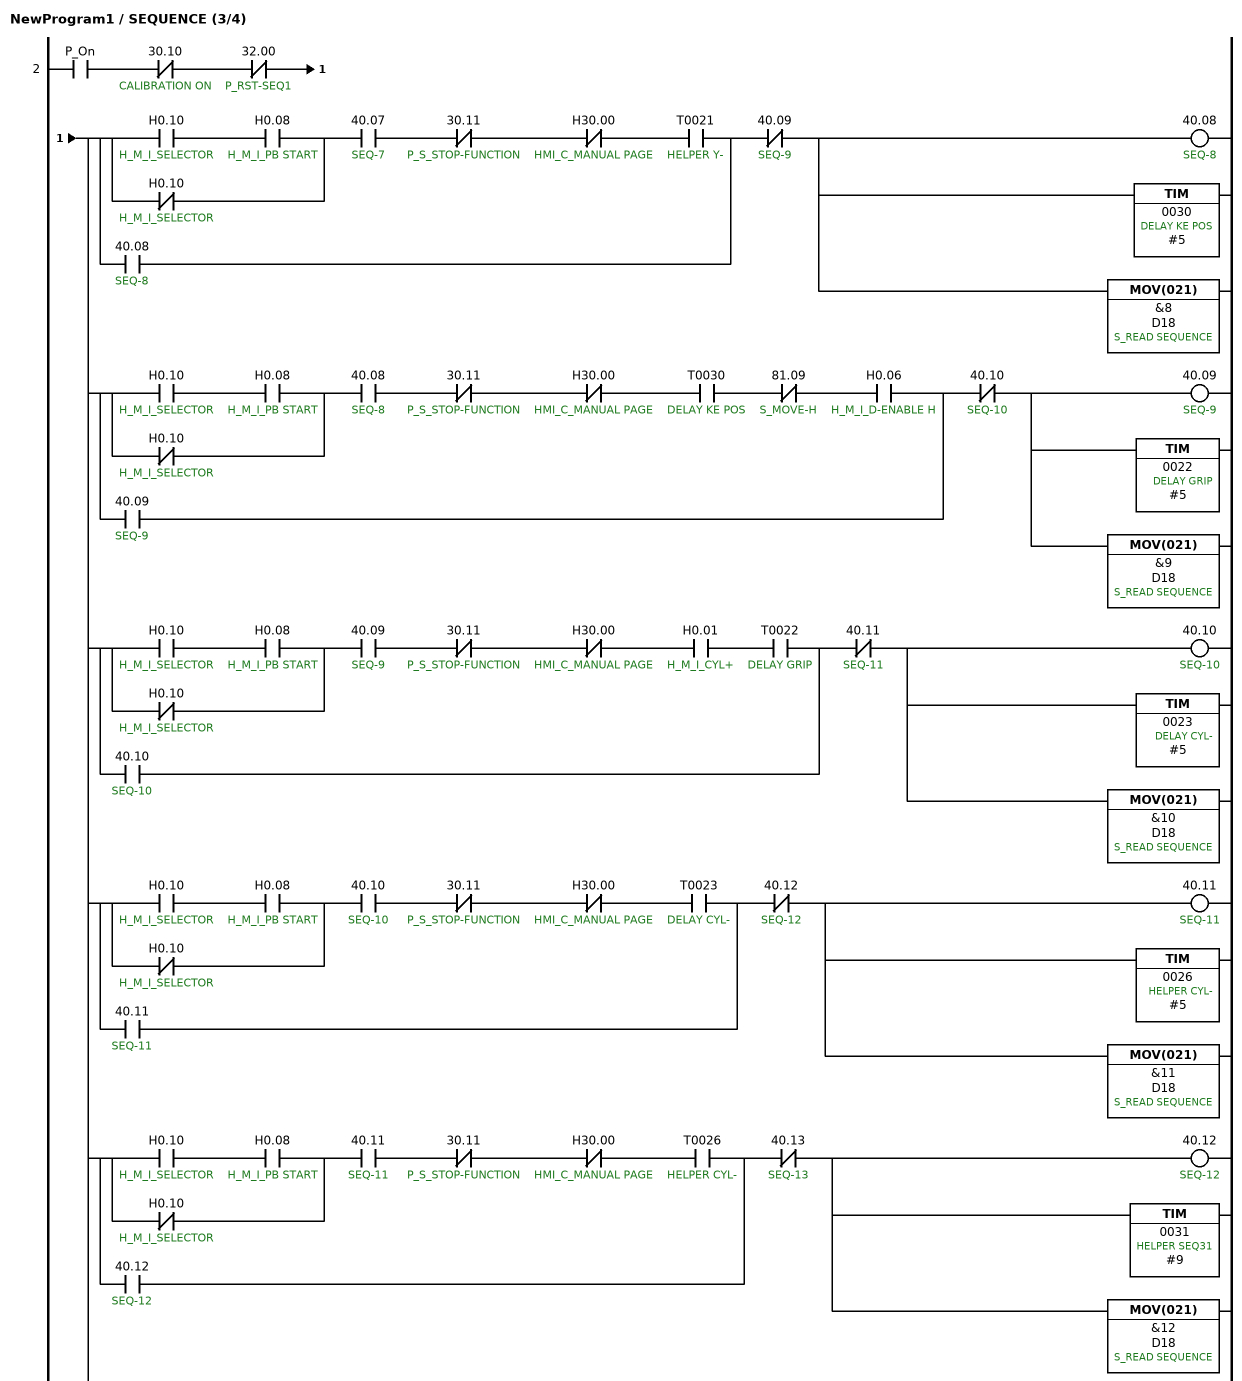

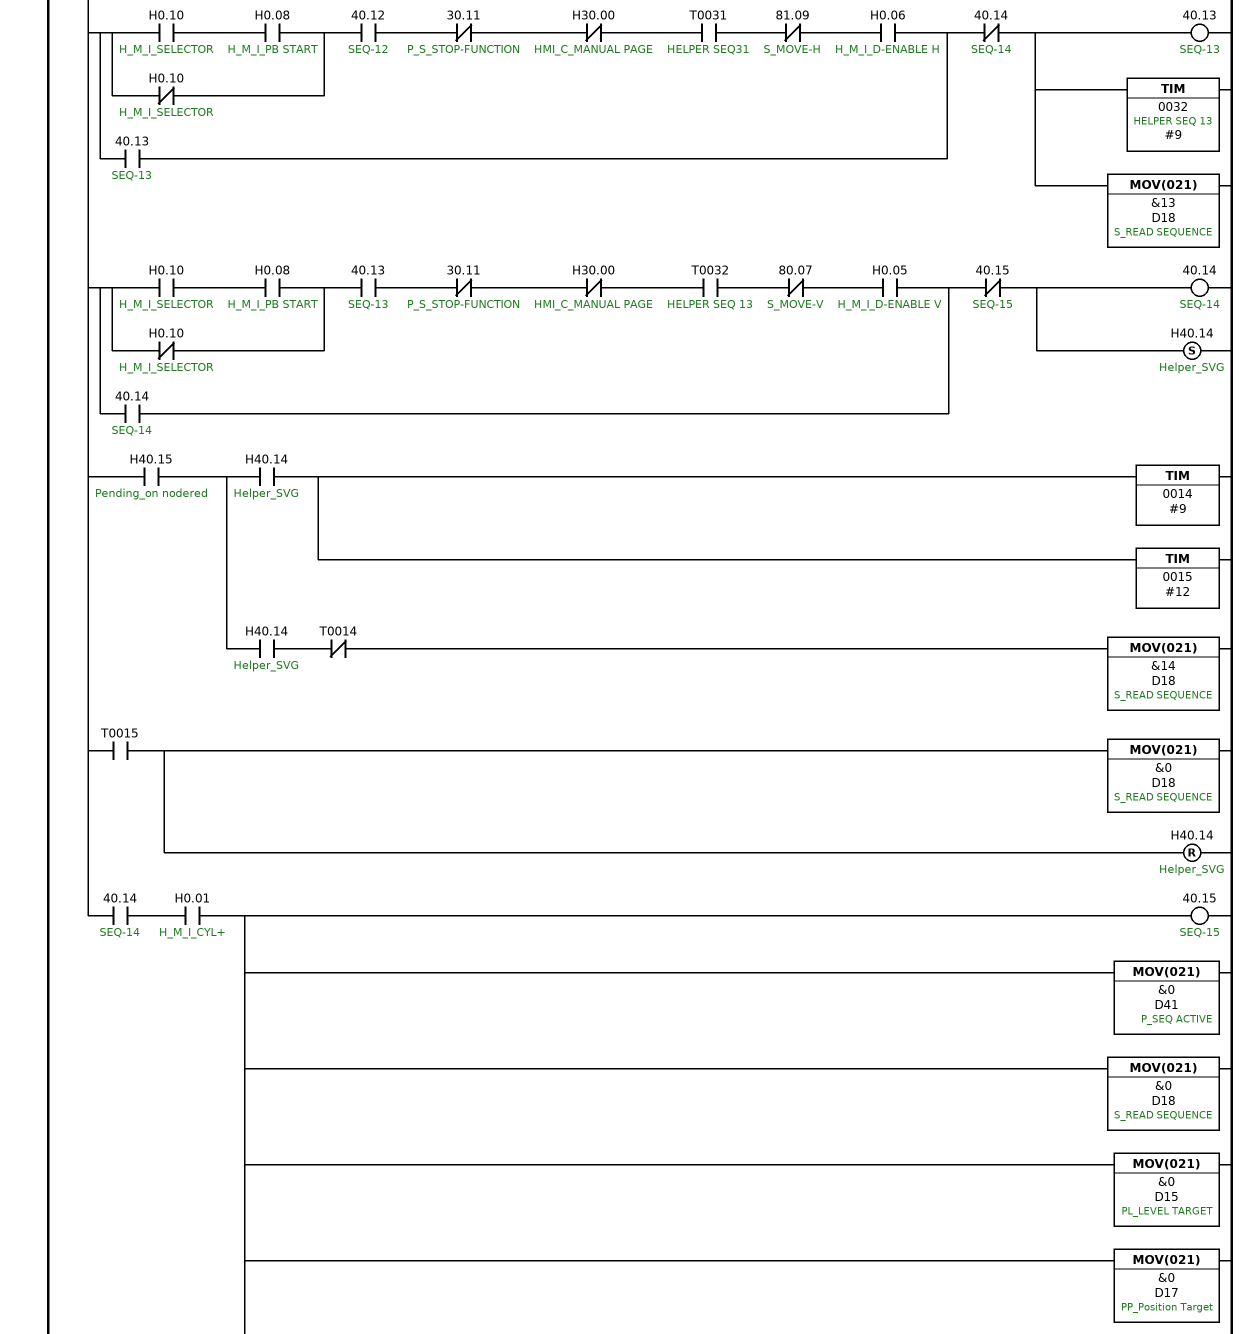

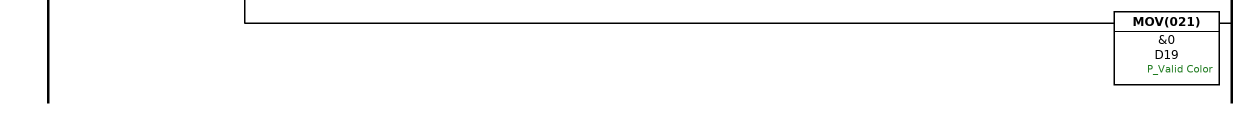
; rung 2
LD P_On
ANDNOT 30.10  ; CALIBRATION ON
ANDNOT 32.00  ; P_RST-SEQ1
OUT TR0
LD H0.10  ; H_M_I_SELECTOR
AND H0.08  ; H_M_I_PB START
ORNOT H0.10  ; H_M_I_SELECTOR
AND 40.07  ; SEQ-7
ANDNOT 30.11  ; P_S_STOP-FUNCTION
ANDNOT H30.00  ; HMI_C_MANUAL PAGE
AND T0021  ; HELPER Y-
OR 40.08  ; SEQ-8
ANDLD
ANDNOT 40.09  ; SEQ-9
OUT 40.08  ; SEQ-8
TIM 0030 #5  ; DELAY KE POS
MOV(021) &8 D18  ; S_READ SEQUENCE
LD TR0
LD H0.10  ; H_M_I_SELECTOR
AND H0.08  ; H_M_I_PB START
ORNOT H0.10  ; H_M_I_SELECTOR
AND 40.08  ; SEQ-8
ANDNOT 30.11  ; P_S_STOP-FUNCTION
ANDNOT H30.00  ; HMI_C_MANUAL PAGE
AND T0030  ; DELAY KE POS
ANDNOT 81.09  ; S_MOVE-H
AND H0.06  ; H_M_I_D-ENABLE H
OR 40.09  ; SEQ-9
ANDLD
ANDNOT 40.10  ; SEQ-10
OUT 40.09  ; SEQ-9
TIM 0022 #5  ; DELAY GRIP
MOV(021) &9 D18  ; S_READ SEQUENCE
LD TR0
LD H0.10  ; H_M_I_SELECTOR
AND H0.08  ; H_M_I_PB START
ORNOT H0.10  ; H_M_I_SELECTOR
AND 40.09  ; SEQ-9
ANDNOT 30.11  ; P_S_STOP-FUNCTION
ANDNOT H30.00  ; HMI_C_MANUAL PAGE
AND H0.01  ; H_M_I_CYL+
AND T0022  ; DELAY GRIP
OR 40.10  ; SEQ-10
ANDLD
ANDNOT 40.11  ; SEQ-11
OUT 40.10  ; SEQ-10
TIM 0023 #5  ; DELAY CYL-
MOV(021) &10 D18  ; S_READ SEQUENCE
LD TR0
LD H0.10  ; H_M_I_SELECTOR
AND H0.08  ; H_M_I_PB START
ORNOT H0.10  ; H_M_I_SELECTOR
AND 40.10  ; SEQ-10
ANDNOT 30.11  ; P_S_STOP-FUNCTION
ANDNOT H30.00  ; HMI_C_MANUAL PAGE
AND T0023  ; DELAY CYL-
OR 40.11  ; SEQ-11
ANDLD
ANDNOT 40.12  ; SEQ-12
OUT 40.11  ; SEQ-11
TIM 0026 #5  ; HELPER CYL-
MOV(021) &11 D18  ; S_READ SEQUENCE
LD TR0
LD H0.10  ; H_M_I_SELECTOR
AND H0.08  ; H_M_I_PB START
ORNOT H0.10  ; H_M_I_SELECTOR
AND 40.11  ; SEQ-11
ANDNOT 30.11  ; P_S_STOP-FUNCTION
ANDNOT H30.00  ; HMI_C_MANUAL PAGE
AND T0026  ; HELPER CYL-
OR 40.12  ; SEQ-12
ANDLD
ANDNOT 40.13  ; SEQ-13
OUT 40.12  ; SEQ-12
TIM 0031 #9  ; HELPER SEQ31
MOV(021) &12 D18  ; S_READ SEQUENCE
LD TR0
LD H0.10  ; H_M_I_SELECTOR
AND H0.08  ; H_M_I_PB START
ORNOT H0.10  ; H_M_I_SELECTOR
AND 40.12  ; SEQ-12
ANDNOT 30.11  ; P_S_STOP-FUNCTION
ANDNOT H30.00  ; HMI_C_MANUAL PAGE
AND T0031  ; HELPER SEQ31
ANDNOT 81.09  ; S_MOVE-H
AND H0.06  ; H_M_I_D-ENABLE H
OR 40.13  ; SEQ-13
ANDLD
ANDNOT 40.14  ; SEQ-14
OUT 40.13  ; SEQ-13
TIM 0032 #9  ; HELPER SEQ 13
MOV(021) &13 D18  ; S_READ SEQUENCE
LD TR0
LD H0.10  ; H_M_I_SELECTOR
AND H0.08  ; H_M_I_PB START
ORNOT H0.10  ; H_M_I_SELECTOR
AND 40.13  ; SEQ-13
ANDNOT 30.11  ; P_S_STOP-FUNCTION
ANDNOT H30.00  ; HMI_C_MANUAL PAGE
AND T0032  ; HELPER SEQ 13
ANDNOT 80.07  ; S_MOVE-V
AND H0.05  ; H_M_I_D-ENABLE V
OR 40.14  ; SEQ-14
ANDLD
ANDNOT 40.15  ; SEQ-15
OUT 40.14  ; SEQ-14
SET H40.14  ; Helper_SVG
LD TR0
AND H40.15  ; Pending_on nodered
OUT TR1
AND H40.14  ; Helper_SVG
TIM 0014 #9
TIM 0015 #12
LD TR1
AND H40.14  ; Helper_SVG
ANDNOT T0014
MOV(021) &14 D18  ; S_READ SEQUENCE
LD TR0
AND T0015
MOV(021) &0 D18  ; S_READ SEQUENCE
RSET H40.14  ; Helper_SVG
LD TR0
AND 40.14  ; SEQ-14
AND H0.01  ; H_M_I_CYL+
OUT 40.15  ; SEQ-15
MOV(021) &0 D41  ; P_SEQ ACTIVE
MOV(021) &0 D18  ; S_READ SEQUENCE
MOV(021) &0 D15  ; PL_LEVEL TARGET
MOV(021) &0 D17  ; PP_Position Target
MOV(021) &0 D19  ; P_Valid Color

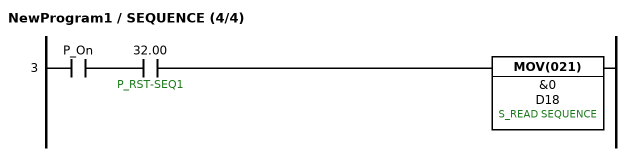
; rung 3
LD P_On
AND 32.00  ; P_RST-SEQ1
MOV(021) &0 D18  ; S_READ SEQUENCE

### Section INPUT

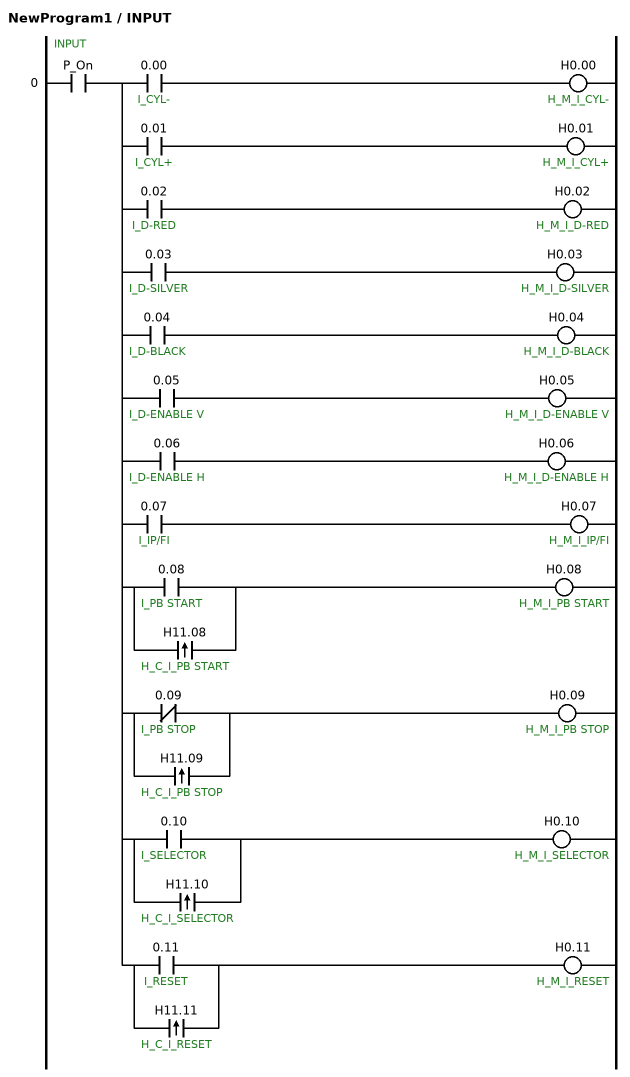
; rung 0: INPUT
LD P_On
OUT TR0
AND 0.00  ; I_CYL-
OUT H0.00  ; H_M_I_CYL-
LD TR0
AND 0.01  ; I_CYL+
OUT H0.01  ; H_M_I_CYL+
LD TR0
AND 0.02  ; I_D-RED
OUT H0.02  ; H_M_I_D-RED
LD TR0
AND 0.03  ; I_D-SILVER
OUT H0.03  ; H_M_I_D-SILVER
LD TR0
AND 0.04  ; I_D-BLACK
OUT H0.04  ; H_M_I_D-BLACK
LD TR0
AND 0.05  ; I_D-ENABLE V
OUT H0.05  ; H_M_I_D-ENABLE V
LD TR0
AND 0.06  ; I_D-ENABLE H
OUT H0.06  ; H_M_I_D-ENABLE H
LD TR0
AND 0.07  ; I_IP/FI
OUT H0.07  ; H_M_I_IP/FI
LD TR0
LD 0.08  ; I_PB START
@OR H11.08  ; H_C_I_PB START
ANDLD
OUT H0.08  ; H_M_I_PB START
LD TR0
LDNOT 0.09  ; I_PB STOP
@OR H11.09  ; H_C_I_PB STOP
ANDLD
OUT H0.09  ; H_M_I_PB STOP
LD TR0
LD 0.10  ; I_SELECTOR
@OR H11.10  ; H_C_I_SELECTOR
ANDLD
OUT H0.10  ; H_M_I_SELECTOR
LD TR0
LD 0.11  ; I_RESET
@OR H11.11  ; H_C_I_RESET
ANDLD
OUT H0.11  ; H_M_I_RESET

### Section OUTPUT

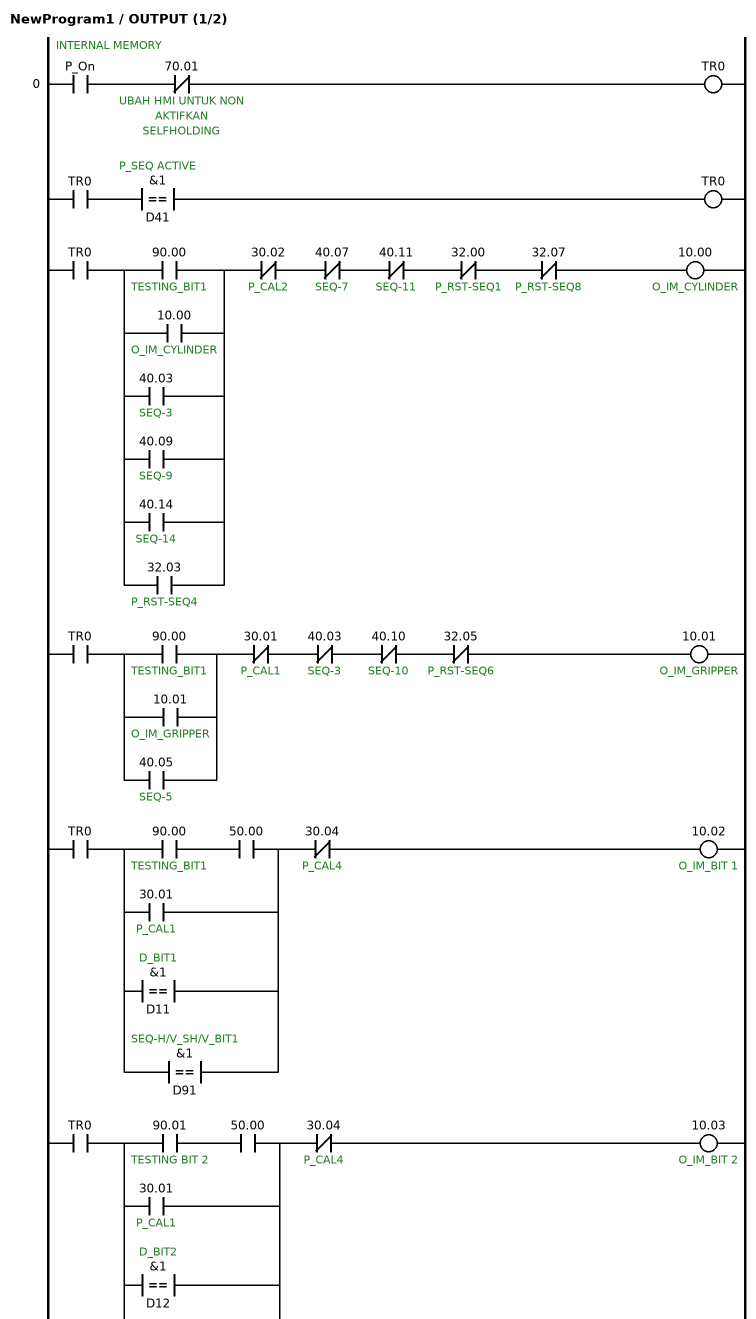

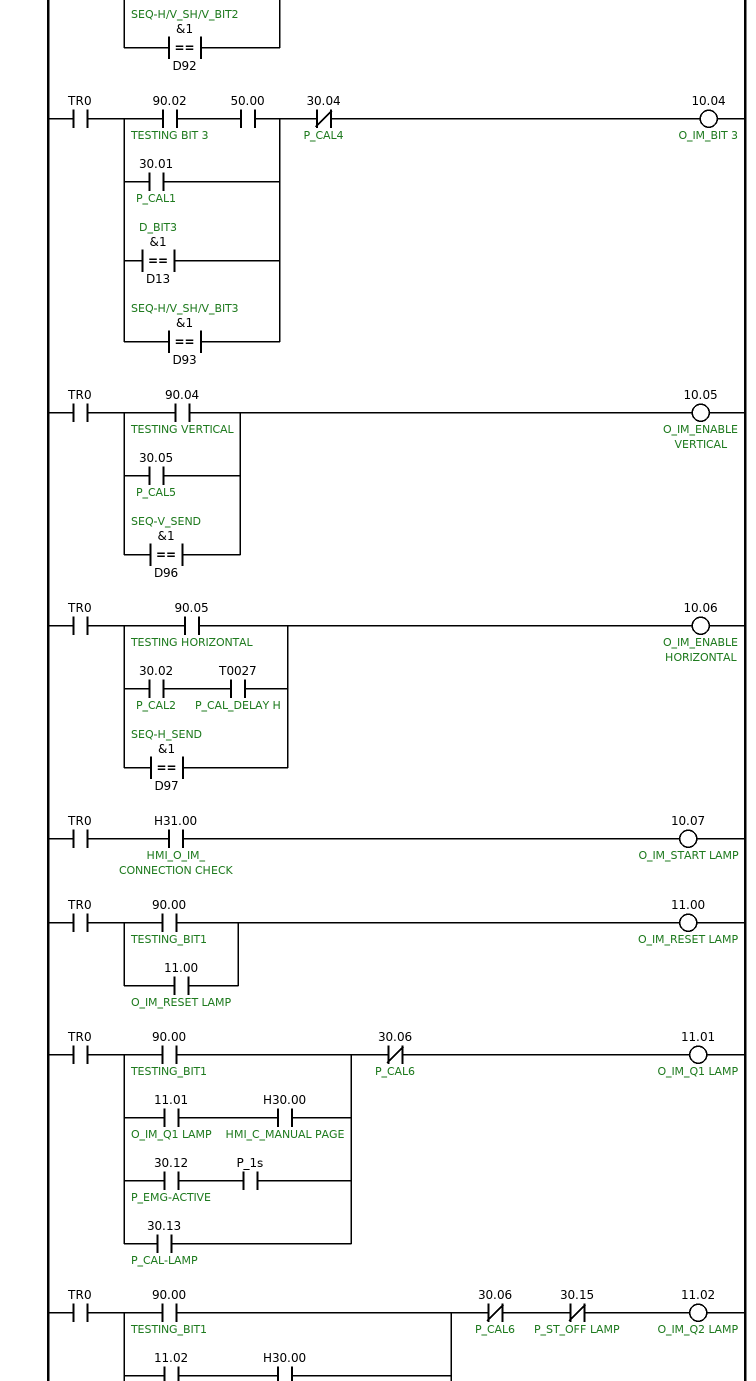

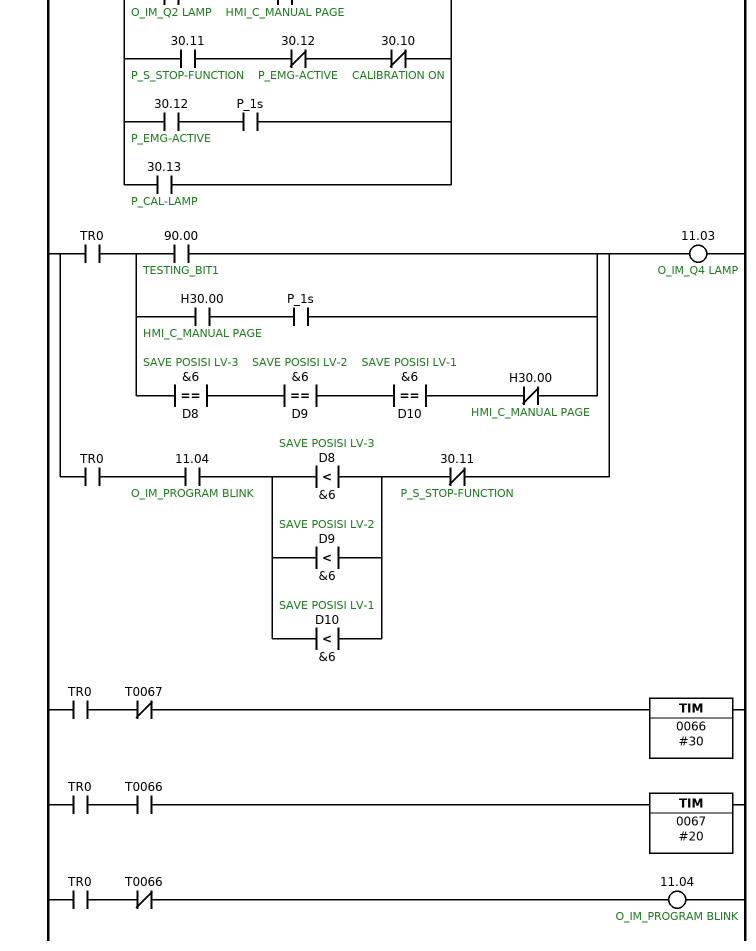
; rung 0: INTERNAL MEMORY
LD P_On
ANDNOT 70.01  ; UBAH HMI UNTUK NON AKTIFKAN SELFHOLDING
OUT TR0
LD 90.00  ; TESTING_BIT1
OR 10.00  ; O_IM_CYLINDER
OR 40.03  ; SEQ-3
OR 40.09  ; SEQ-9
OR 40.14  ; SEQ-14
OR 32.03  ; P_RST-SEQ4
ANDLD
ANDNOT 30.02  ; P_CAL2
ANDNOT 40.07  ; SEQ-7
ANDNOT 40.11  ; SEQ-11
ANDNOT 32.00  ; P_RST-SEQ1
ANDNOT 32.07  ; P_RST-SEQ8
OUT 10.00  ; O_IM_CYLINDER
LD TR0
LD 90.00  ; TESTING_BIT1
OR 10.01  ; O_IM_GRIPPER
OR 40.05  ; SEQ-5
ANDLD
ANDNOT 30.01  ; P_CAL1
ANDNOT 40.03  ; SEQ-3
ANDNOT 40.10  ; SEQ-10
ANDNOT 32.05  ; P_RST-SEQ6
OUT 10.01  ; O_IM_GRIPPER
LD TR0
LD 90.00  ; TESTING_BIT1
AND 50.00
OR 30.01  ; P_CAL1
OR=(300) &1 D11  ; D_BIT1
OR=(300) &1 D91  ; SEQ-H/V_SH/V_BIT1
ANDLD
ANDNOT 30.04  ; P_CAL4
OUT 10.02  ; O_IM_BIT 1
LD TR0
LD 90.01  ; TESTING BIT 2
AND 50.00
OR 30.01  ; P_CAL1
OR=(300) &1 D12  ; D_BIT2
OR=(300) &1 D92  ; SEQ-H/V_SH/V_BIT2
ANDLD
ANDNOT 30.04  ; P_CAL4
OUT 10.03  ; O_IM_BIT 2
LD TR0
LD 90.02  ; TESTING BIT 3
AND 50.00
OR 30.01  ; P_CAL1
OR=(300) &1 D13  ; D_BIT3
OR=(300) &1 D93  ; SEQ-H/V_SH/V_BIT3
ANDLD
ANDNOT 30.04  ; P_CAL4
OUT 10.04  ; O_IM_BIT 3
LD TR0
LD 90.04  ; TESTING VERTICAL
OR 30.05  ; P_CAL5
OR=(300) &1 D96  ; SEQ-V_SEND
ANDLD
OUT 10.05  ; O_IM_ENABLE VERTICAL
LD TR0
LD 90.05  ; TESTING HORIZONTAL
LD 30.02  ; P_CAL2
AND T0027  ; P_CAL_DELAY H
ORLD
OR=(300) &1 D97  ; SEQ-H_SEND
ANDLD
OUT 10.06  ; O_IM_ENABLE HORIZONTAL
LD TR0
AND H31.00  ; HMI_O_IM_CONNECTION CHECK
OUT 10.07  ; O_IM_START LAMP
LD TR0
LD 90.00  ; TESTING_BIT1
OR 11.00  ; O_IM_RESET LAMP
ANDLD
OUT 11.00  ; O_IM_RESET LAMP
LD TR0
LD 90.00  ; TESTING_BIT1
LD 11.01  ; O_IM_Q1 LAMP
AND H30.00  ; HMI_C_MANUAL PAGE
ORLD
LD 30.12  ; P_EMG-ACTIVE
AND P_1s
ORLD
OR 30.13  ; P_CAL-LAMP
ANDLD
ANDNOT 30.06  ; P_CAL6
OUT 11.01  ; O_IM_Q1 LAMP
LD TR0
LD 90.00  ; TESTING_BIT1
LD 11.02  ; O_IM_Q2 LAMP
AND H30.00  ; HMI_C_MANUAL PAGE
ORLD
LD 30.11  ; P_S_STOP-FUNCTION
ANDNOT 30.12  ; P_EMG-ACTIVE
ANDNOT 30.10  ; CALIBRATION ON
ORLD
LD 30.12  ; P_EMG-ACTIVE
AND P_1s
ORLD
OR 30.13  ; P_CAL-LAMP
ANDLD
ANDNOT 30.06  ; P_CAL6
ANDNOT 30.15  ; P_ST_OFF LAMP
OUT 11.02  ; O_IM_Q2 LAMP
LD TR0
LD 90.00  ; TESTING_BIT1
LD H30.00  ; HMI_C_MANUAL PAGE
AND P_1s
ORLD
LD=(300) &6 D8  ; SAVE POSISI LV-3
AND=(300) &6 D9  ; SAVE POSISI LV-2
AND=(300) &6 D10  ; SAVE POSISI LV-1
ANDNOT H30.00  ; HMI_C_MANUAL PAGE
ORLD
ANDLD
LD TR0
AND=(300) &1 D41  ; P_SEQ ACTIVE
OUT TR0
AND 11.04  ; O_IM_PROGRAM BLINK
LD<(310) D8 &6  ; SAVE POSISI LV-3
OR<(310) D9 &6  ; SAVE POSISI LV-2
OR<(310) D10 &6  ; SAVE POSISI LV-1
ANDLD
ANDNOT 30.11  ; P_S_STOP-FUNCTION
ORLD
OUT 11.03  ; O_IM_Q4 LAMP
LD TR0
ANDNOT T0067
TIM 0066 #30
LD TR0
AND T0066
TIM 0067 #20
LD TR0
ANDNOT T0066
OUT 11.04  ; O_IM_PROGRAM BLINK

